FUNCTION_BLOCK FB_MoveAbsoluteNC IMPLEMENTS I_MoveAbsolute
VAR
    {attribute 'no_copy'}
    AxisRef : REFERENCE TO AXIS_REF;
    // MoveABsolute
    fbMcMoveAbsolute : MC_MoveAbsolute;
    fTargetPosition	: LREAL;
    fTargetVelocity	: LREAL;
    fTargetAcceleration	: LREAL := 0.0;
    fTargetDeceleration	: LREAL := 0.0;
    fTargetJerk	: LREAL := 0.0;
    eBufferMode	: MC_BufferMode := MC_BufferMode.MC_Aborting;
    rtBusy : R_TRIG;
    ftBusy : F_TRIG;
    rtDone : R_TRIG;
    rtAborted : R_TRIG;
    bCommandMoveAbsolute : BOOL;
    bAborted : BOOL;
    bError : BOOL;
    bBusy : BOOL;
    bDone : BOOL;
    bActive : BOOL;
    nErrorID : UDINT;
    sMessage : T_MAXSTRING;
END_VAR

THIS^.AxisRef.ReadStatus();

THIS^.fbMcMoveAbsolute(
    Axis := THIS^.AxisRef,
    Execute := THIS^.bCommandMoveAbsolute,
    Position := THIS^.fTargetPosition,
    Velocity := THIS^.fTargetVelocity,
    Acceleration := THIS^.fTargetAcceleration,
    Deceleration := THIS^.fTargetDeceleration,
    Jerk := THIS^.fTargetJerk,
    BufferMode := THIS^.eBufferMode,
    Done => ,
    Busy => THIS^.bBusy,
    Active => ,
    CommandAborted => THIS^.bAborted,
    Error => THIS^.bError,
    ErrorID => THIS^.nErrorID
);

rtBusy (CLK:=bBusy);
ftBusy(CLK:=bBusy);
// to be checked
bDone S= ftBusy.Q AND NOT THIS^.bError AND NOT THIS^.AxisRef.Status.HasJob;
bDone R= rtBusy.Q;

// Reset execute after when done successfull or after abort reset
// this way the done and error condition is latched till next move or global reset.
rtDone(CLK:=bDone);
rtAborted(CLK:=bAborted);
IF  rtDone.Q OR rtAborted.Q THEN
    THIS^.bCommandMoveAbsolute := FALSE;
END_IF

{warning 'Add property implementation'}
PROPERTY Aborted : BOOL
GET
Aborted := THIS^.bAborted;
END_GET
END_PROPERTY

{warning 'Add property implementation'}
PROPERTY Active : BOOL
GET
Active := bActive;
END_GET
END_PROPERTY

{warning 'add property implementation'}
PROPERTY Busy : BOOL
GET
Busy := THIS^.bBusy;
END_GET
END_PROPERTY

METHOD PUBLIC CallAfterInit
VAR_INPUT
	AxisRef : REFERENCE TO AXIS_REF;
END_VAR
THIS^.AxisRef REF= AxisRef;
END_METHOD

PROPERTY CommandMoveAbsolute : BOOL
SET
bCommandMoveAbsolute := CommandMoveAbsolute;
END_SET
END_PROPERTY

{warning 'add property implementation'}
PROPERTY Done : BOOL
GET
Done := THIS^.bDone;
END_GET
END_PROPERTY

{warning 'add property implementation'}
PROPERTY Error : BOOL
GET
Error := THIS^.bError;
END_GET
END_PROPERTY

{warning 'add property implementation'}
PROPERTY ErrorID : UDINT
GET
ErrorID := THIS^.nErrorID;
END_GET
END_PROPERTY

METHOD FB_Init : BOOL
VAR_INPUT
    bInitRetains : BOOL; // if TRUE, the retain variables are initialized (warm start / cold start)
    bInCopyCode : BOOL;  // if TRUE, the instance afterwards gets moved into the copy code (online change)
    AxisRef : REFERENCE TO AXIS_REF;
END_VAR
THIS^.AxisRef REF= AxisRef;
END_METHOD

PROPERTY Message : T_MAXSTRING
GET
Message := sMessage;
END_GET
END_PROPERTY

METHOD MoveAbsolute
VAR_INPUT
    Execute     : BOOL;
    Position	: LREAL;
    Velocity	: LREAL;
    Acceleration	: LREAL := 0.0;
    Deceleration	: LREAL := 0.0;
    Jerk	: LREAL := 0.0;
    BufferMode	: MC_BufferMode := MC_BufferMode.MC_Aborting;
END_VAR
THIS^.bCommandMoveAbsolute := Execute;
THIS^.fTargetPosition := Position;
THIS^.fTargetVelocity := Velocity;
THIS^.fTargetAcceleration := Acceleration;
THIS^.fTargetDeceleration := Deceleration;
THIS^.fTargetJerk := Jerk;
THIS^.eBufferMode := BufferMode;
END_METHOD

END_FUNCTION_BLOCK

(* stored: Version 1.1.0.1
   POU FB_MoveAbsoluteNC: Id {e71196e8-5955-4e1c-a924-f415b73d00ec}, SpecialFunc None
   Property Aborted: Id {e282a52e-140a-4032-b49e-bebd36434e55}
   Get Get: Id {d29e9ff4-92f9-427a-9ec7-fa6fbbe474b3}
   Property Active: Id {dd75b655-9142-4732-8a04-757a4f64e51a}
   Get Get: Id {a477c2f4-fc88-4b80-b4f4-7805da1fb7a8}
   Property Busy: Id {1ae87be5-03cb-4a25-b603-7a901b104320}
   Get Get: Id {9d197ce2-8fd9-4bc1-99a9-01c16a01edb5}
   Method CallAfterInit: Id {00377abf-4ca1-4aa0-a1c2-987e6f8750e8}
   Property CommandMoveAbsolute: Id {7bbe24c9-46f3-48a9-9a5a-f238ba708042}
   Set Set: Id {5ca86cbe-838d-4ff0-b334-f0d7b6e6a752}
   Property Done: Id {a764e9fb-e6d3-4787-bb5e-f18a571f3537}
   Get Get: Id {50c96990-1ca2-4598-9b3c-4ce1d489107b}
   Property Error: Id {0185f2b2-2e6f-442f-b749-2bbd8da7d055}
   Get Get: Id {1e0b343f-fb19-4817-9dd8-a79547d284ae}
   Property ErrorID: Id {765d4df4-ef37-4baf-a5b2-0caf395dd3d5}
   Get Get: Id {616d42e5-15ca-457d-9573-bf6beb7c1f43}
   Method FB_Init: Id {e87d7c58-75a2-4628-877e-343a902489c2}
   Property Message: Id {13938688-fe04-4182-8021-54fdd58e055d}
   Get Get: Id {59125684-2209-4efb-a11e-261b597d4642}
   Method MoveAbsolute: Id {ec9e8694-906a-4f94-b53d-2b2ff2681c1a} *)
